Staubli VAL3: loadJoint.pgx

public program loadJoint(string x_sItem, num& x_nResult)
  local string l_sType
  local string l_sMessage
  local num l_nResult
begin
  //
  // !!! REMOVE DUE PROBLEMS of CROSS LINK
  //
  //
  //  // load the select trajectory..already loaded
  //  call getTrajType(l_sType)
  //  if find(jPoint:libPath(),saveData:sPathTraj)==-1
  //    l_nResult=jPoint:libLoad(saveData:sPathTraj+"JPOINT")
  //    delay(0)
  //    if saveData:bDebug
  //      ? "HOME loading JPOINT..."+saveData:sPathTraj+"JPOINT"+toString("",l_nResult)
  //    endIf
  //  endIf
  //  if isDefined(jPoint:tTraj[x_sItem])
  //    // validate
  //    x_nResult=0
  //  elseIf x_sItem!=""
  //    // not FOUND
  //    call language:message(l_sMessage,-7)
  //    x_nResult=-1
  //    popUpMsg(l_sMessage+x_sItem)
  //  endIf
end
